Yaskawa INFORM job: TEST-MACRO.JBI

/JOB
//NAME TEST-MACRO
//POS
///NPOS 0,0,0,0,0,0
//INST
///DATE 2018/11/14 10:50
///ATTR SC,RW
///GROUP1 RB1,BS1
NOP
MACRO1 MJ#(0) ARGF5
END
